// TIA Portal V16 export
// export: Created 2020-05-27T18:57:34.0416305Z, ExportSetting None, DisplayName Totally Integrated Automation Portal, DisplayVersion V16 Update 1, DisplayName TIA Portal Version Control Interface, DisplayVersion V16, DisplayName TIA Portal Openness, DisplayVersion V16 Update 1, DisplayName SINAMICS Startdrive Advanced, DisplayVersion V16 Update 2, DisplayName SINAMICS Startdrive G130, G150, S120, S150, SINAMICS MV, S210, DisplayVersion V16 Update 2, DisplayName SINAMICS Startdrive G110M, G120, G120C, G120D, G120P, DisplayVersion V16 Update 2, DisplayName STEP 7 Professional, DisplayVersion V16 Update 1, DisplayName STEP 7 Safety, DisplayVersion V16, DisplayName WinCC Advanced, DisplayVersion V16 Update 1
FUNCTION_BLOCK "Block_Logic"   // FB1, LAD
{ S7_Optimized_Access := 'TRUE' }
// stored: MemoryReserve 100, SetENOAutomatically false
   VAR_INPUT
      A1 : Bool;
   END_VAR
   VAR_OUTPUT
      Out1 : Bool;
   END_VAR
   VAR_TEMP
      MyValue : Bool;
   END_VAR
BEGIN

REGION Network 1
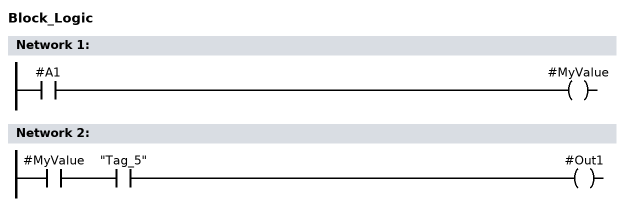
   RUNG wire#powerrail
      Contact( #A1 )
      Coil( #MyValue )
   END_RUNG
   // the same network as SCL:
   #MyValue := #A1;
END_REGION

REGION Network 2
   RUNG wire#powerrail
      Contact( #MyValue )
      Contact( "Tag_5" )
      Coil( #Out1 )
   END_RUNG
   // the same network as SCL:
   #Out1 := #MyValue AND "Tag_5";
END_REGION
END_FUNCTION_BLOCK
